FUNCTION_BLOCK ABSTRACT FiberSwitchBase EXTENDS TExecution IMPLEMENTS IDevice
VAR_INPUT
END_VAR
VAR_OUTPUT
END_VAR
VAR
	{attribute 'OPC.UA.DA' := '0'}
	_name : STRING;
	{attribute 'OPC.UA.DA' := '0'}
	_deviceID : STRING;					
	{attribute 'OPC.UA.DA' := '0'}
	_family : DeviceFamily;	
	{attribute 'OPC.UA.DA' := '0'}	
	_logger : Logger;
	{attribute 'OPC.UA.DA' := '0'}
	_message : StringBuilder;
	{attribute 'OPC.UA.DA' := '0'}
	_fiberSwitchConfig : DeviceConfiguration;
END_VAR

METHOD PROTECTED ABSTRACT CurrentPosition
VAR_INPUT
	Execute : BOOL;
END_VAR
END_METHOD

PROPERTY DeviceID : STRING
GET
DeviceID := _deviceID;
END_GET
SET
_deviceID := DeviceID;
END_SET
END_PROPERTY

PROPERTY Family : DeviceFamily
GET
Family := _family;
END_GET
SET
_family := Family;
END_SET
END_PROPERTY

PROPERTY Name : STRING
GET
Name := _name;
END_GET
SET
_name := Name;
END_SET
END_PROPERTY

METHOD PROTECTED ABSTRACT SetSwitchPosition
VAR_INPUT
	Execute : BOOL;
	Position : UINT;
END_VAR
END_METHOD

END_FUNCTION_BLOCK

(* stored: Version 1.1.0.1, ProductVersion 3.1.4024.3
   POU FiberSwitchBase: Id {be951fd9-6127-43c7-bbfa-faa7db4fe84f}, SpecialFunc None
   Method CurrentPosition: Id {11876318-5d79-46a0-b8ae-16aadabbab6a}
   Property DeviceID: Id {f8ddf66d-3cfb-4601-9f17-73dfa2f86187}
   Get Get: Id {dff0611c-3bc4-40ab-bc9e-138120ffe139}
   Set Set: Id {e50f8f62-6fea-43d2-a3f6-c93f36e1d56b}
   Property Family: Id {c475aa4d-516b-4e82-a450-d4625bb5fe5a}
   Get Get: Id {d3f7b0bb-1853-4de2-89fc-194c24e0eaae}
   Set Set: Id {436ae111-271f-4cf3-ab9c-f33a0c1fc50e}
   Property Name: Id {2d432f9e-4454-4561-b86c-a4b4ac8dfed8}
   Get Get: Id {dda8e867-cd38-4524-9577-d4514de55745}
   Set Set: Id {942370ad-debf-4ddf-83ae-a1e4d4e13b46}
   Method SetSwitchPosition: Id {53bd3248-99fe-40ce-a488-2be7e1f9540c} *)
